{attribute addProperty BoxType "AT2050-0501-0024"}
{attribute addProperty Id "A_0084_AT2050_5500_0017_AT2050_5500AT2050_3DCFC8D064080"}
{attribute addProperty CRC "1420891119"}
{attribute addProperty SizeInBites "640"}
{attribute addProperty SizeInBytes "80"}
TYPE A_0072_AT2050_0501_0024_AT2050_0501_54B113EF EXTENDS AT2050_9506A482 :
STRUCT
	{attribute addProperty Name "A_0084_AT2050_5500_0017_AT2050_5500"}
	A_0084_AT2050_5500_0017_AT2050_5500 : AT2050_3DCFC8D0;
END_STRUCT
END_TYPE

(* stored: Version 1.2.0.0, ProductVersion 3.1.4024.9
   DUT A_0072_AT2050_0501_0024_AT2050_0501_54B113EF: Id {3c84b949-2720-41b5-b2c8-a90b2c306895} *)
